FUNCTION Convert_DATE_TO_ULINT : Hresult
VAR_INPUT
	in : DATE;
	out : REFERENCE TO ULINT;
END_VAR
VAR
	converted : ULINT;
END_VAR

converted := DATE_TO_ULINT(in);

IF (ULINT_TO_DATE(converted) <> in) THEN
	Convert_DATE_TO_ULINT := INCOMPATIBLE;
	RETURN;
END_IF

out := converted;

END_FUNCTION

(* stored: Version 1.1.0.1, ProductVersion 3.1.4024.12
   POU Convert_DATE_TO_ULINT: Id {4f4405e9-edf5-494b-9ad2-f0c9776609a8}, SpecialFunc None *)
